(* PLC project io_engine_2d2s, Dassault Systèmes ControlBuild 2024x *)
(* stored: creationDateTime 2023-10-03T11:12:47-01:00 *)

PROGRAM panel
  VAR_OUTPUT
    forwardPB : BOOL := false;
    backwardPB : BOOL := false;
    highSpeedPB : BOOL := false;
    lowSpeedPB : BOOL := false;
    stopPB : BOOL := false;
  END_VAR

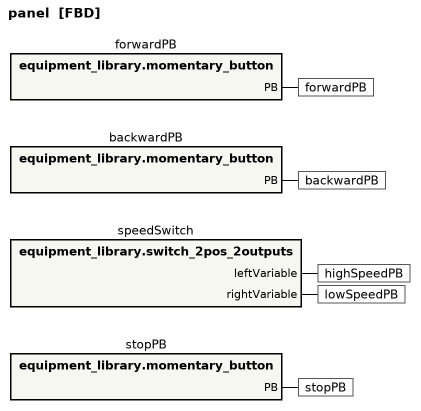
(* FBD diagram, written out as Structured Text *)
forwardPB();
forwardPB := forwardPB.PB;
backwardPB();
backwardPB := backwardPB.PB;
speedSwitch();
highSpeedPB := speedSwitch.leftVariable;
lowSpeedPB := speedSwitch.rightVariable;
stopPB();
stopPB := stopPB.PB;
END_PROGRAM

(* Integrated object C/C+OP of a motor with two speed and two directions *)
PROGRAM io_library.io_engine_2d2s
  VAR_INPUT
    autoMode : BOOL := false;
    manualMode : BOOL := false;
  END_VAR
  VAR_INPUT
    autoFwdCmd : BOOL := false;
    autoBwdCmd : BOOL := false;
    autoHSCmd : BOOL := false;
    autoLSCmd : BOOL := false;
  END_VAR
  VAR_INPUT
    acknowledgePB : BOOL := false;
  END_VAR
  VAR_OUTPUT
    speedVal : REAL := 0.0;
    speedPercent : REAL := 0.0;
  END_VAR
  VAR_OUTPUT
    generalFault : BOOL := false;
  END_VAR

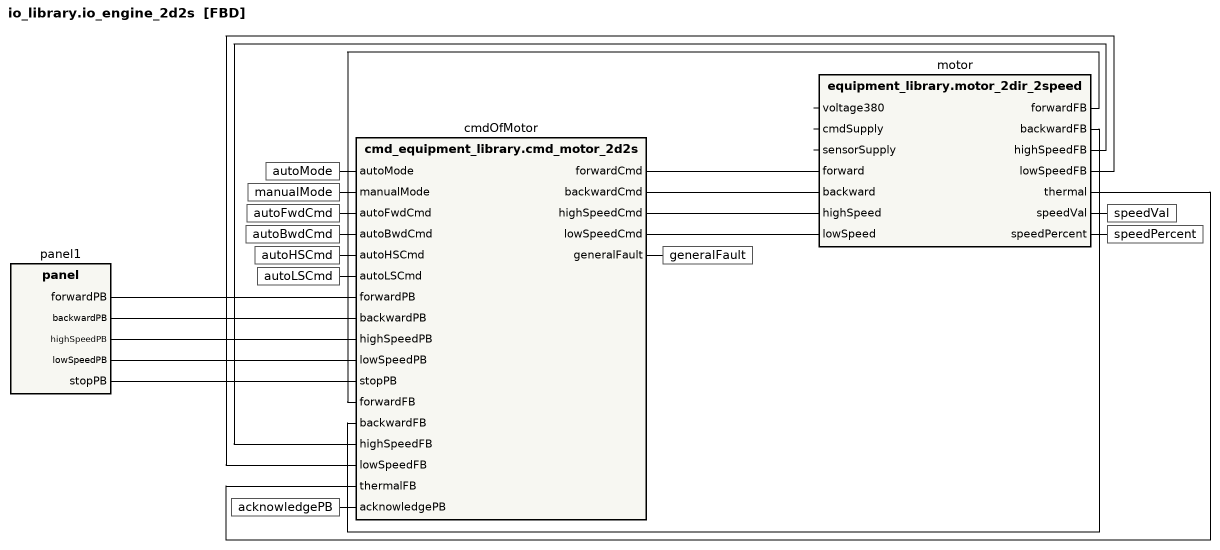
(* FBD diagram, written out as Structured Text *)
panel1();
motor(forward := cmdOfMotor.forwardCmd, backward := cmdOfMotor.backwardCmd, highSpeed := cmdOfMotor.highSpeedCmd, lowSpeed := cmdOfMotor.lowSpeedCmd);
cmdOfMotor(autoMode := autoMode, manualMode := manualMode, autoFwdCmd := autoFwdCmd, autoBwdCmd := autoBwdCmd, autoHSCmd := autoHSCmd, autoLSCmd := autoLSCmd, forwardPB := panel1.forwardPB, backwardPB := panel1.backwardPB, highSpeedPB := panel1.highSpeedPB, lowSpeedPB := panel1.lowSpeedPB, stopPB := panel1.stopPB, forwardFB := motor.forwardFB, backwardFB := motor.backwardFB, highSpeedFB := motor.highSpeedFB, lowSpeedFB := motor.lowSpeedFB, thermalFB := motor.thermal, acknowledgePB := acknowledgePB);
generalFault := cmdOfMotor.generalFault;
speedVal := motor.speedVal;
speedPercent := motor.speedPercent;
END_PROGRAM
